FUNCTION_BLOCK FB_LamparaAsignada_LD
// La lampara se enciende mientras se acciona el pulsador
VAR
    Lampara   AT %Q*  : BOOL;
    Pulsador  AT %I*  : BOOL;
END_VAR

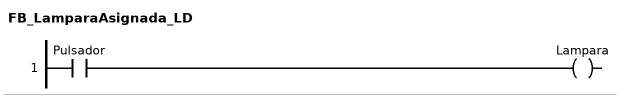
// NETWORK 1
Lampara := Pulsador;

END_FUNCTION_BLOCK

(* stored: Version 1.1.0.1, ProductVersion 3.1.4024.15
   POU FB_LamparaAsignada_LD: Id {e94e976e-ba2a-4361-86cb-52f381bc806b}, SpecialFunc None *)
